{attribute 'pack_mode' := '2'}
TYPE ST_R_ProgParameter :
STRUCT
  _nStart               : DINT := 900;
  _nCount               : DINT := 10;
  _rRParamsWrite        : ARRAY[0..MAX_R_PARA] OF LREAL;
  _rRParamsRead         : ARRAY[0..MAX_R_PARA] OF LREAL;
END_STRUCT
END_TYPE

(* stored: Version 1.1.0.1, ProductVersion 3.1.4024.12
   DUT ST_R_ProgParameter: Id {b16fac44-2267-02bd-3dff-41ed6e746315} *)
